(*
SPDX-FileCopyrightText: © 2026 Oleksandr Tiutyk <trofimich@gmail.com>
SPDX-License-Identifier: MIT
License: https://opensource.org/license/mit
*)

(*!
<summary>Common object metadata and identity. Interface references do not transfer ownership.</summary>
<description>
Members require a live instance; they cannot validate an object after its lifetime has ended.
</description>
*)

INTERFACE IObject EXTENDS __SYSTEM.IQueryInterface

(*!
<summary>Borrowed reference to class-name storage, not an independent string copy.</summary>
*)

{attribute 'monitoring' := 'call'}

PROPERTY ClassName : REFERENCE TO STRING
GET
END_GET
END_PROPERTY

(*!
<summary>Object compares instance identity by default; a derived implementation may override this method.</summary>
*)

{attribute "object_name" := "Equals"}

METHOD Equals : BOOL
VAR_INPUT 
	object : IObject;
END_VAR
END_METHOD

(*!
<summary>Returns the namespace-qualified type name by value, within the return string capacity.</summary>
*)

METHOD GetFullTypeName : STRING
END_METHOD

(*!
<summary>Returns a diagnostic object name by value; it is not a unique object identifier.</summary>
*)

METHOD GetName : WSTRING
VAR_INPUT
END_VAR
END_METHOD

(*!
<summary>Reports the memory area, not ownership or registration for automatic cleanup.</summary>
*)

{attribute 'monitoring' := 'call'}

PROPERTY FINAL IsDynamicInstance : BOOL
GET
END_GET
END_PROPERTY

(*!
<summary>Borrowed reference to namespace-name storage, not an independent string copy.</summary>
*)

{attribute 'monitoring' := 'call'}

PROPERTY NamespaceName : REFERENCE TO STRING
GET
END_GET
END_PROPERTY

(*!
<summary>Borrowed address of this instance. Obtaining it does not grant permission to delete the object.</summary>
*)

{attribute 'monitoring' := 'call'}

PROPERTY SelfAddress : POINTER TO Object
GET
END_GET
END_PROPERTY

(*!
<summary>Size in bytes of the complete concrete instance; excludes separately allocated buffers it owns.</summary>
*)

{attribute 'monitoring' := 'call'}

PROPERTY SelfSize : ULINT
GET
END_GET
END_PROPERTY

END_INTERFACE

(* stored: Version 1.1.0.1
   Itf IObject: Id {ead88c25-62c0-46e5-b40b-3c9531c283b1}
   Property ClassName: Id {3e7a3cd3-d8e0-4d8a-8c55-1b5342aa67c1}
   Get Get: Id {889c3d50-a912-431d-828b-b0aa9026a512}
   Method Equals: Id {1d3007f2-f5ed-4237-a812-4ec6c04abeaf}
   Method GetFullTypeName: Id {5fd27adb-4d7b-498f-9cad-32d06a6d8894}
   Method GetName: Id {8294dede-68ca-42ff-a38b-cc86adf90d8b}
   Property IsDynamicInstance: Id {46fa710c-bc2b-4e4c-a911-56db473aa5ff}
   Get Get: Id {e52ef2de-1fe8-4d12-944f-685b8a1320b6}
   Property NamespaceName: Id {41a2bdb9-dadd-4c91-851c-acf2ad853661}
   Get Get: Id {415a0a62-f677-4d44-b3ed-d7eb98e6d4aa}
   Property SelfAddress: Id {6b5d769e-7b05-4a19-a56c-3656121e0615}
   Get Get: Id {22ecdebc-d7a0-45cc-9cfa-c59fbc5dff05}
   Property SelfSize: Id {902a9b17-518a-4f74-97b7-bd1998b63b8c}
   Get Get: Id {6b36f7ed-1855-4e40-a186-1ed3287e25da} *)
